Fanuc KAREL source: kb00035.KL

-- PROVISIONAL review KL for V940-1; original PC SHA256 fe7c27902b29e3096d90944d94660ab283946edc3e6979b5a36723ddb583811b
-- Incomplete behavior may be omitted. Consult companion uncertainty JSON. Do not deploy.
PROGRAM KB00035
%NOLOCKGROUP
BEGIN
  -- V9_ZERO_TABLE_METADATA_HINT layout=0002_ascii; no indexed target words; source/name/runtime held
  -- UNRESOLVED_PC offsets 5-12; opcodes 9D,23
  -- UNRESOLVED_PC offsets 17-24; opcodes 9D,23
  -- UNRESOLVED_PC offsets 29-36; opcodes 9D,23
  -- UNRESOLVED_PC offsets 41-50; opcodes 3F,75
  -- UNRESOLVED_PC offsets 55-85; opcodes 27,22,22,22,22,2A,31
  -- UNRESOLVED_PC offsets 90-94; opcodes 7F
END KB00035
